// TIA Portal V18 export
// export: Created 2026-01-09T11:31:57.3502958Z, ExportSetting WithDefaults, DisplayName Totally Integrated Automation Portal, DisplayVersion V18 Update 5, DisplayName TIA Portal Openness, DisplayVersion V18 Update 5, DisplayName TIA Portal Teamcenter Gateway, DisplayVersion V18, DisplayName TIA Portal Version Control Interface, DisplayVersion V18, DisplayName SINAMICS Startdrive Advanced, DisplayVersion V18 SP2 Update 1, DisplayName SINAMICS Startdrive G110M, G120, G120C, G120D, G120P, G115D, DisplayVersion V18 SP2 Update 1, DisplayName SINAMICS Startdrive G130, G150, S120, S150, SINAMICS MV, S210, G220, S200, DisplayVersion V18 SP2 Update 1, DisplayName STEP 7 Professional, DisplayVersion V18 Update 5, DisplayName STEP 7 Safety, DisplayVersion V18, DisplayName WinCC Professional, DisplayVersion V18 Update 5
TagTable "Axis"
  Parameter_AxisRun_Axis{1} : ServoType_UDT  (PLC tag Parameter.AxisRun.Axis[1], CPU S71500-2PN_TP700, 1 s)
    TagStructureMember "Pos1"
      TagStructureMember "Position"
      TagStructureMember "Speed"
      TagStructureMember "Reached"
    TagStructureMember "Pos2"
      TagStructureMember "Position"
      TagStructureMember "Speed"
      TagStructureMember "Reached"
    TagStructureMember "Pos3"
      TagStructureMember "Position"
      TagStructureMember "Speed"
      TagStructureMember "Reached"
    TagStructureMember "Pos4"
      TagStructureMember "Position"
      TagStructureMember "Speed"
      TagStructureMember "Reached"
    TagStructureMember "Pos5"
      TagStructureMember "Position"
      TagStructureMember "Speed"
      TagStructureMember "Reached"
    TagStructureMember "Pos6"
      TagStructureMember "Position"
      TagStructureMember "Speed"
      TagStructureMember "Reached"
    TagStructureMember "Pos7"
      TagStructureMember "Position"
      TagStructureMember "Speed"
      TagStructureMember "Reached"
    TagStructureMember "Pos8"
      TagStructureMember "Position"
      TagStructureMember "Speed"
      TagStructureMember "Reached"
    TagStructureMember "Pos9"
      TagStructureMember "Position"
      TagStructureMember "Speed"
      TagStructureMember "Reached"
    TagStructureMember "Pos10"
      TagStructureMember "Position"
      TagStructureMember "Speed"
      TagStructureMember "Reached"
    TagStructureMember "Pos11"
      TagStructureMember "Position"
      TagStructureMember "Speed"
      TagStructureMember "Reached"
    TagStructureMember "Pos12"
      TagStructureMember "Position"
      TagStructureMember "Speed"
      TagStructureMember "Reached"
    TagStructureMember "Pos13"
      TagStructureMember "Position"
      TagStructureMember "Speed"
      TagStructureMember "Reached"
    TagStructureMember "Pos14"
      TagStructureMember "Position"
      TagStructureMember "Speed"
      TagStructureMember "Reached"
    TagStructureMember "Pos15"
      TagStructureMember "Position"
      TagStructureMember "Speed"
      TagStructureMember "Reached"
    TagStructureMember "Pos16"
      TagStructureMember "Position"
      TagStructureMember "Speed"
      TagStructureMember "Reached"
    TagStructureMember "Pos17"
      TagStructureMember "Position"
      TagStructureMember "Speed"
      TagStructureMember "Reached"
    TagStructureMember "Pos18"
      TagStructureMember "Position"
      TagStructureMember "Speed"
      TagStructureMember "Reached"
    TagStructureMember "Pos19"
      TagStructureMember "Position"
      TagStructureMember "Speed"
      TagStructureMember "Reached"
    TagStructureMember "Pos20"
      TagStructureMember "Position"
      TagStructureMember "Speed"
      TagStructureMember "Reached"
    TagStructureMember "Pos21"
      TagStructureMember "Position"
      TagStructureMember "Speed"
      TagStructureMember "Reached"
    TagStructureMember "Pos22"
      TagStructureMember "Position"
      TagStructureMember "Speed"
      TagStructureMember "Reached"
    TagStructureMember "Pos23"
      TagStructureMember "Position"
      TagStructureMember "Speed"
      TagStructureMember "Reached"
    TagStructureMember "Pos24"
      TagStructureMember "Position"
      TagStructureMember "Speed"
      TagStructureMember "Reached"
    TagStructureMember "Pos25"
      TagStructureMember "Position"
      TagStructureMember "Speed"
      TagStructureMember "Reached"
    TagStructureMember "Pos26"
      TagStructureMember "Position"
      TagStructureMember "Speed"
      TagStructureMember "Reached"
    TagStructureMember "Pos27"
      TagStructureMember "Position"
      TagStructureMember "Speed"
      TagStructureMember "Reached"
    TagStructureMember "Pos28"
      TagStructureMember "Position"
      TagStructureMember "Speed"
      TagStructureMember "Reached"
    TagStructureMember "Pos29"
      TagStructureMember "Position"
      TagStructureMember "Speed"
      TagStructureMember "Reached"
    TagStructureMember "Pos30"
      TagStructureMember "Position"
      TagStructureMember "Speed"
      TagStructureMember "Reached"
  Parameter_AxisRun_Axis{2} : ServoType_UDT  (PLC tag Parameter.AxisRun.Axis[2], CPU S71500-2PN_TP700, 1 s)
    TagStructureMember "Pos1"
      TagStructureMember "Position"
      TagStructureMember "Speed"
      TagStructureMember "Reached"
    TagStructureMember "Pos2"
      TagStructureMember "Position"
      TagStructureMember "Speed"
      TagStructureMember "Reached"
    TagStructureMember "Pos3"
      TagStructureMember "Position"
      TagStructureMember "Speed"
      TagStructureMember "Reached"
    TagStructureMember "Pos4"
      TagStructureMember "Position"
      TagStructureMember "Speed"
      TagStructureMember "Reached"
    TagStructureMember "Pos5"
      TagStructureMember "Position"
      TagStructureMember "Speed"
      TagStructureMember "Reached"
    TagStructureMember "Pos6"
      TagStructureMember "Position"
      TagStructureMember "Speed"
      TagStructureMember "Reached"
    TagStructureMember "Pos7"
      TagStructureMember "Position"
      TagStructureMember "Speed"
      TagStructureMember "Reached"
    TagStructureMember "Pos8"
      TagStructureMember "Position"
      TagStructureMember "Speed"
      TagStructureMember "Reached"
    TagStructureMember "Pos9"
      TagStructureMember "Position"
      TagStructureMember "Speed"
      TagStructureMember "Reached"
    TagStructureMember "Pos10"
      TagStructureMember "Position"
      TagStructureMember "Speed"
      TagStructureMember "Reached"
    TagStructureMember "Pos11"
      TagStructureMember "Position"
      TagStructureMember "Speed"
      TagStructureMember "Reached"
    TagStructureMember "Pos12"
      TagStructureMember "Position"
      TagStructureMember "Speed"
      TagStructureMember "Reached"
    TagStructureMember "Pos13"
      TagStructureMember "Position"
      TagStructureMember "Speed"
      TagStructureMember "Reached"
    TagStructureMember "Pos14"
      TagStructureMember "Position"
      TagStructureMember "Speed"
      TagStructureMember "Reached"
    TagStructureMember "Pos15"
      TagStructureMember "Position"
      TagStructureMember "Speed"
      TagStructureMember "Reached"
    TagStructureMember "Pos16"
      TagStructureMember "Position"
      TagStructureMember "Speed"
      TagStructureMember "Reached"
    TagStructureMember "Pos17"
      TagStructureMember "Position"
      TagStructureMember "Speed"
      TagStructureMember "Reached"
    TagStructureMember "Pos18"
      TagStructureMember "Position"
      TagStructureMember "Speed"
      TagStructureMember "Reached"
    TagStructureMember "Pos19"
      TagStructureMember "Position"
      TagStructureMember "Speed"
      TagStructureMember "Reached"
    TagStructureMember "Pos20"
      TagStructureMember "Position"
      TagStructureMember "Speed"
      TagStructureMember "Reached"
    TagStructureMember "Pos21"
      TagStructureMember "Position"
      TagStructureMember "Speed"
      TagStructureMember "Reached"
    TagStructureMember "Pos22"
      TagStructureMember "Position"
      TagStructureMember "Speed"
      TagStructureMember "Reached"
    TagStructureMember "Pos23"
      TagStructureMember "Position"
      TagStructureMember "Speed"
      TagStructureMember "Reached"
    TagStructureMember "Pos24"
      TagStructureMember "Position"
      TagStructureMember "Speed"
      TagStructureMember "Reached"
    TagStructureMember "Pos25"
      TagStructureMember "Position"
      TagStructureMember "Speed"
      TagStructureMember "Reached"
    TagStructureMember "Pos26"
      TagStructureMember "Position"
      TagStructureMember "Speed"
      TagStructureMember "Reached"
    TagStructureMember "Pos27"
      TagStructureMember "Position"
      TagStructureMember "Speed"
      TagStructureMember "Reached"
    TagStructureMember "Pos28"
      TagStructureMember "Position"
      TagStructureMember "Speed"
      TagStructureMember "Reached"
    TagStructureMember "Pos29"
      TagStructureMember "Position"
      TagStructureMember "Speed"
      TagStructureMember "Reached"
    TagStructureMember "Pos30"
      TagStructureMember "Position"
      TagStructureMember "Speed"
      TagStructureMember "Reached"
  Parameter_AxisRun_Axis{3} : ServoType_UDT  (PLC tag Parameter.AxisRun.Axis[3], CPU S71500-2PN_TP700, 1 s)
    TagStructureMember "Pos1"
      TagStructureMember "Position"
      TagStructureMember "Speed"
      TagStructureMember "Reached"
    TagStructureMember "Pos2"
      TagStructureMember "Position"
      TagStructureMember "Speed"
      TagStructureMember "Reached"
    TagStructureMember "Pos3"
      TagStructureMember "Position"
      TagStructureMember "Speed"
      TagStructureMember "Reached"
    TagStructureMember "Pos4"
      TagStructureMember "Position"
      TagStructureMember "Speed"
      TagStructureMember "Reached"
    TagStructureMember "Pos5"
      TagStructureMember "Position"
      TagStructureMember "Speed"
      TagStructureMember "Reached"
    TagStructureMember "Pos6"
      TagStructureMember "Position"
      TagStructureMember "Speed"
      TagStructureMember "Reached"
    TagStructureMember "Pos7"
      TagStructureMember "Position"
      TagStructureMember "Speed"
      TagStructureMember "Reached"
    TagStructureMember "Pos8"
      TagStructureMember "Position"
      TagStructureMember "Speed"
      TagStructureMember "Reached"
    TagStructureMember "Pos9"
      TagStructureMember "Position"
      TagStructureMember "Speed"
      TagStructureMember "Reached"
    TagStructureMember "Pos10"
      TagStructureMember "Position"
      TagStructureMember "Speed"
      TagStructureMember "Reached"
    TagStructureMember "Pos11"
      TagStructureMember "Position"
      TagStructureMember "Speed"
      TagStructureMember "Reached"
    TagStructureMember "Pos12"
      TagStructureMember "Position"
      TagStructureMember "Speed"
      TagStructureMember "Reached"
    TagStructureMember "Pos13"
      TagStructureMember "Position"
      TagStructureMember "Speed"
      TagStructureMember "Reached"
    TagStructureMember "Pos14"
      TagStructureMember "Position"
      TagStructureMember "Speed"
      TagStructureMember "Reached"
    TagStructureMember "Pos15"
      TagStructureMember "Position"
      TagStructureMember "Speed"
      TagStructureMember "Reached"
    TagStructureMember "Pos16"
      TagStructureMember "Position"
      TagStructureMember "Speed"
      TagStructureMember "Reached"
    TagStructureMember "Pos17"
      TagStructureMember "Position"
      TagStructureMember "Speed"
      TagStructureMember "Reached"
    TagStructureMember "Pos18"
      TagStructureMember "Position"
      TagStructureMember "Speed"
      TagStructureMember "Reached"
    TagStructureMember "Pos19"
      TagStructureMember "Position"
      TagStructureMember "Speed"
      TagStructureMember "Reached"
    TagStructureMember "Pos20"
      TagStructureMember "Position"
      TagStructureMember "Speed"
      TagStructureMember "Reached"
    TagStructureMember "Pos21"
      TagStructureMember "Position"
      TagStructureMember "Speed"
      TagStructureMember "Reached"
    TagStructureMember "Pos22"
      TagStructureMember "Position"
      TagStructureMember "Speed"
      TagStructureMember "Reached"
    TagStructureMember "Pos23"
      TagStructureMember "Position"
      TagStructureMember "Speed"
      TagStructureMember "Reached"
    TagStructureMember "Pos24"
      TagStructureMember "Position"
      TagStructureMember "Speed"
      TagStructureMember "Reached"
    TagStructureMember "Pos25"
      TagStructureMember "Position"
      TagStructureMember "Speed"
      TagStructureMember "Reached"
    TagStructureMember "Pos26"
      TagStructureMember "Position"
      TagStructureMember "Speed"
      TagStructureMember "Reached"
    TagStructureMember "Pos27"
      TagStructureMember "Position"
      TagStructureMember "Speed"
      TagStructureMember "Reached"
    TagStructureMember "Pos28"
      TagStructureMember "Position"
      TagStructureMember "Speed"
      TagStructureMember "Reached"
    TagStructureMember "Pos29"
      TagStructureMember "Position"
      TagStructureMember "Speed"
      TagStructureMember "Reached"
    TagStructureMember "Pos30"
      TagStructureMember "Position"
      TagStructureMember "Speed"
      TagStructureMember "Reached"
  Parameter_AxisRun_Axis{4} : ServoType_UDT  (PLC tag Parameter.AxisRun.Axis[4], CPU S71500-2PN_TP700, 1 s)
    TagStructureMember "Pos1"
      TagStructureMember "Position"
      TagStructureMember "Speed"
      TagStructureMember "Reached"
    TagStructureMember "Pos2"
      TagStructureMember "Position"
      TagStructureMember "Speed"
      TagStructureMember "Reached"
    TagStructureMember "Pos3"
      TagStructureMember "Position"
      TagStructureMember "Speed"
      TagStructureMember "Reached"
    TagStructureMember "Pos4"
      TagStructureMember "Position"
      TagStructureMember "Speed"
      TagStructureMember "Reached"
    TagStructureMember "Pos5"
      TagStructureMember "Position"
      TagStructureMember "Speed"
      TagStructureMember "Reached"
    TagStructureMember "Pos6"
      TagStructureMember "Position"
      TagStructureMember "Speed"
      TagStructureMember "Reached"
    TagStructureMember "Pos7"
      TagStructureMember "Position"
      TagStructureMember "Speed"
      TagStructureMember "Reached"
    TagStructureMember "Pos8"
      TagStructureMember "Position"
      TagStructureMember "Speed"
      TagStructureMember "Reached"
    TagStructureMember "Pos9"
      TagStructureMember "Position"
      TagStructureMember "Speed"
      TagStructureMember "Reached"
    TagStructureMember "Pos10"
      TagStructureMember "Position"
      TagStructureMember "Speed"
      TagStructureMember "Reached"
    TagStructureMember "Pos11"
      TagStructureMember "Position"
      TagStructureMember "Speed"
      TagStructureMember "Reached"
    TagStructureMember "Pos12"
      TagStructureMember "Position"
      TagStructureMember "Speed"
      TagStructureMember "Reached"
    TagStructureMember "Pos13"
      TagStructureMember "Position"
      TagStructureMember "Speed"
      TagStructureMember "Reached"
    TagStructureMember "Pos14"
      TagStructureMember "Position"
      TagStructureMember "Speed"
      TagStructureMember "Reached"
    TagStructureMember "Pos15"
      TagStructureMember "Position"
      TagStructureMember "Speed"
      TagStructureMember "Reached"
    TagStructureMember "Pos16"
      TagStructureMember "Position"
      TagStructureMember "Speed"
      TagStructureMember "Reached"
    TagStructureMember "Pos17"
      TagStructureMember "Position"
      TagStructureMember "Speed"
      TagStructureMember "Reached"
    TagStructureMember "Pos18"
      TagStructureMember "Position"
      TagStructureMember "Speed"
      TagStructureMember "Reached"
    TagStructureMember "Pos19"
      TagStructureMember "Position"
      TagStructureMember "Speed"
      TagStructureMember "Reached"
    TagStructureMember "Pos20"
      TagStructureMember "Position"
      TagStructureMember "Speed"
      TagStructureMember "Reached"
    TagStructureMember "Pos21"
      TagStructureMember "Position"
      TagStructureMember "Speed"
      TagStructureMember "Reached"
    TagStructureMember "Pos22"
      TagStructureMember "Position"
      TagStructureMember "Speed"
      TagStructureMember "Reached"
    TagStructureMember "Pos23"
      TagStructureMember "Position"
      TagStructureMember "Speed"
      TagStructureMember "Reached"
    TagStructureMember "Pos24"
      TagStructureMember "Position"
      TagStructureMember "Speed"
      TagStructureMember "Reached"
    TagStructureMember "Pos25"
      TagStructureMember "Position"
      TagStructureMember "Speed"
      TagStructureMember "Reached"
    TagStructureMember "Pos26"
      TagStructureMember "Position"
      TagStructureMember "Speed"
      TagStructureMember "Reached"
    TagStructureMember "Pos27"
      TagStructureMember "Position"
      TagStructureMember "Speed"
      TagStructureMember "Reached"
    TagStructureMember "Pos28"
      TagStructureMember "Position"
      TagStructureMember "Speed"
      TagStructureMember "Reached"
    TagStructureMember "Pos29"
      TagStructureMember "Position"
      TagStructureMember "Speed"
      TagStructureMember "Reached"
    TagStructureMember "Pos30"
      TagStructureMember "Position"
      TagStructureMember "Speed"
      TagStructureMember "Reached"
  Parameter_AxisRun_Axis{5} : ServoType_UDT  (PLC tag Parameter.AxisRun.Axis[5], CPU S71500-2PN_TP700, 1 s)
    TagStructureMember "Pos1"
      TagStructureMember "Position"
      TagStructureMember "Speed"
      TagStructureMember "Reached"
    TagStructureMember "Pos2"
      TagStructureMember "Position"
      TagStructureMember "Speed"
      TagStructureMember "Reached"
    TagStructureMember "Pos3"
      TagStructureMember "Position"
      TagStructureMember "Speed"
      TagStructureMember "Reached"
    TagStructureMember "Pos4"
      TagStructureMember "Position"
      TagStructureMember "Speed"
      TagStructureMember "Reached"
    TagStructureMember "Pos5"
      TagStructureMember "Position"
      TagStructureMember "Speed"
      TagStructureMember "Reached"
    TagStructureMember "Pos6"
      TagStructureMember "Position"
      TagStructureMember "Speed"
      TagStructureMember "Reached"
    TagStructureMember "Pos7"
      TagStructureMember "Position"
      TagStructureMember "Speed"
      TagStructureMember "Reached"
    TagStructureMember "Pos8"
      TagStructureMember "Position"
      TagStructureMember "Speed"
      TagStructureMember "Reached"
    TagStructureMember "Pos9"
      TagStructureMember "Position"
      TagStructureMember "Speed"
      TagStructureMember "Reached"
    TagStructureMember "Pos10"
      TagStructureMember "Position"
      TagStructureMember "Speed"
      TagStructureMember "Reached"
    TagStructureMember "Pos11"
      TagStructureMember "Position"
      TagStructureMember "Speed"
      TagStructureMember "Reached"
    TagStructureMember "Pos12"
      TagStructureMember "Position"
      TagStructureMember "Speed"
      TagStructureMember "Reached"
    TagStructureMember "Pos13"
      TagStructureMember "Position"
      TagStructureMember "Speed"
      TagStructureMember "Reached"
    TagStructureMember "Pos14"
      TagStructureMember "Position"
      TagStructureMember "Speed"
      TagStructureMember "Reached"
    TagStructureMember "Pos15"
      TagStructureMember "Position"
      TagStructureMember "Speed"
      TagStructureMember "Reached"
    TagStructureMember "Pos16"
      TagStructureMember "Position"
      TagStructureMember "Speed"
      TagStructureMember "Reached"
    TagStructureMember "Pos17"
      TagStructureMember "Position"
      TagStructureMember "Speed"
      TagStructureMember "Reached"
    TagStructureMember "Pos18"
      TagStructureMember "Position"
      TagStructureMember "Speed"
      TagStructureMember "Reached"
    TagStructureMember "Pos19"
      TagStructureMember "Position"
      TagStructureMember "Speed"
      TagStructureMember "Reached"
    TagStructureMember "Pos20"
      TagStructureMember "Position"
      TagStructureMember "Speed"
      TagStructureMember "Reached"
    TagStructureMember "Pos21"
      TagStructureMember "Position"
      TagStructureMember "Speed"
      TagStructureMember "Reached"
    TagStructureMember "Pos22"
      TagStructureMember "Position"
      TagStructureMember "Speed"
      TagStructureMember "Reached"
    TagStructureMember "Pos23"
      TagStructureMember "Position"
      TagStructureMember "Speed"
      TagStructureMember "Reached"
    TagStructureMember "Pos24"
      TagStructureMember "Position"
      TagStructureMember "Speed"
      TagStructureMember "Reached"
    TagStructureMember "Pos25"
      TagStructureMember "Position"
      TagStructureMember "Speed"
      TagStructureMember "Reached"
    TagStructureMember "Pos26"
      TagStructureMember "Position"
      TagStructureMember "Speed"
      TagStructureMember "Reached"
    TagStructureMember "Pos27"
      TagStructureMember "Position"
      TagStructureMember "Speed"
      TagStructureMember "Reached"
    TagStructureMember "Pos28"
      TagStructureMember "Position"
      TagStructureMember "Speed"
      TagStructureMember "Reached"
    TagStructureMember "Pos29"
      TagStructureMember "Position"
      TagStructureMember "Speed"
      TagStructureMember "Reached"
    TagStructureMember "Pos30"
      TagStructureMember "Position"
      TagStructureMember "Speed"
      TagStructureMember "Reached"
  Parameter_AxisRun_Axis{6} : ServoType_UDT  (PLC tag Parameter.AxisRun.Axis[6], CPU S71500-2PN_TP700, 1 s)
    TagStructureMember "Pos1"
      TagStructureMember "Position"
      TagStructureMember "Speed"
      TagStructureMember "Reached"
    TagStructureMember "Pos2"
      TagStructureMember "Position"
      TagStructureMember "Speed"
      TagStructureMember "Reached"
    TagStructureMember "Pos3"
      TagStructureMember "Position"
      TagStructureMember "Speed"
      TagStructureMember "Reached"
    TagStructureMember "Pos4"
      TagStructureMember "Position"
      TagStructureMember "Speed"
      TagStructureMember "Reached"
    TagStructureMember "Pos5"
      TagStructureMember "Position"
      TagStructureMember "Speed"
      TagStructureMember "Reached"
    TagStructureMember "Pos6"
      TagStructureMember "Position"
      TagStructureMember "Speed"
      TagStructureMember "Reached"
    TagStructureMember "Pos7"
      TagStructureMember "Position"
      TagStructureMember "Speed"
      TagStructureMember "Reached"
    TagStructureMember "Pos8"
      TagStructureMember "Position"
      TagStructureMember "Speed"
      TagStructureMember "Reached"
    TagStructureMember "Pos9"
      TagStructureMember "Position"
      TagStructureMember "Speed"
      TagStructureMember "Reached"
    TagStructureMember "Pos10"
      TagStructureMember "Position"
      TagStructureMember "Speed"
      TagStructureMember "Reached"
    TagStructureMember "Pos11"
      TagStructureMember "Position"
      TagStructureMember "Speed"
      TagStructureMember "Reached"
    TagStructureMember "Pos12"
      TagStructureMember "Position"
      TagStructureMember "Speed"
      TagStructureMember "Reached"
    TagStructureMember "Pos13"
      TagStructureMember "Position"
      TagStructureMember "Speed"
      TagStructureMember "Reached"
    TagStructureMember "Pos14"
      TagStructureMember "Position"
      TagStructureMember "Speed"
      TagStructureMember "Reached"
    TagStructureMember "Pos15"
      TagStructureMember "Position"
      TagStructureMember "Speed"
      TagStructureMember "Reached"
    TagStructureMember "Pos16"
      TagStructureMember "Position"
      TagStructureMember "Speed"
      TagStructureMember "Reached"
    TagStructureMember "Pos17"
      TagStructureMember "Position"
      TagStructureMember "Speed"
      TagStructureMember "Reached"
    TagStructureMember "Pos18"
      TagStructureMember "Position"
      TagStructureMember "Speed"
      TagStructureMember "Reached"
    TagStructureMember "Pos19"
      TagStructureMember "Position"
      TagStructureMember "Speed"
      TagStructureMember "Reached"
    TagStructureMember "Pos20"
      TagStructureMember "Position"
      TagStructureMember "Speed"
      TagStructureMember "Reached"
    TagStructureMember "Pos21"
      TagStructureMember "Position"
      TagStructureMember "Speed"
      TagStructureMember "Reached"
    TagStructureMember "Pos22"
      TagStructureMember "Position"
      TagStructureMember "Speed"
      TagStructureMember "Reached"
    TagStructureMember "Pos23"
      TagStructureMember "Position"
      TagStructureMember "Speed"
      TagStructureMember "Reached"
    TagStructureMember "Pos24"
      TagStructureMember "Position"
      TagStructureMember "Speed"
      TagStructureMember "Reached"
    TagStructureMember "Pos25"
      TagStructureMember "Position"
      TagStructureMember "Speed"
      TagStructureMember "Reached"
    TagStructureMember "Pos26"
      TagStructureMember "Position"
      TagStructureMember "Speed"
      TagStructureMember "Reached"
    TagStructureMember "Pos27"
      TagStructureMember "Position"
      TagStructureMember "Speed"
      TagStructureMember "Reached"
    TagStructureMember "Pos28"
      TagStructureMember "Position"
      TagStructureMember "Speed"
      TagStructureMember "Reached"
    TagStructureMember "Pos29"
      TagStructureMember "Position"
      TagStructureMember "Speed"
      TagStructureMember "Reached"
    TagStructureMember "Pos30"
      TagStructureMember "Position"
      TagStructureMember "Speed"
      TagStructureMember "Reached"
  Parameter_AxisRun_Axis{7} : ServoType_UDT  (PLC tag Parameter.AxisRun.Axis[7], CPU S71500-2PN_TP700, 1 s)
    TagStructureMember "Pos1"
      TagStructureMember "Position"
      TagStructureMember "Speed"
      TagStructureMember "Reached"
    TagStructureMember "Pos2"
      TagStructureMember "Position"
      TagStructureMember "Speed"
      TagStructureMember "Reached"
    TagStructureMember "Pos3"
      TagStructureMember "Position"
      TagStructureMember "Speed"
      TagStructureMember "Reached"
    TagStructureMember "Pos4"
      TagStructureMember "Position"
      TagStructureMember "Speed"
      TagStructureMember "Reached"
    TagStructureMember "Pos5"
      TagStructureMember "Position"
      TagStructureMember "Speed"
      TagStructureMember "Reached"
    TagStructureMember "Pos6"
      TagStructureMember "Position"
      TagStructureMember "Speed"
      TagStructureMember "Reached"
    TagStructureMember "Pos7"
      TagStructureMember "Position"
      TagStructureMember "Speed"
      TagStructureMember "Reached"
    TagStructureMember "Pos8"
      TagStructureMember "Position"
      TagStructureMember "Speed"
      TagStructureMember "Reached"
    TagStructureMember "Pos9"
      TagStructureMember "Position"
      TagStructureMember "Speed"
      TagStructureMember "Reached"
    TagStructureMember "Pos10"
      TagStructureMember "Position"
      TagStructureMember "Speed"
      TagStructureMember "Reached"
    TagStructureMember "Pos11"
      TagStructureMember "Position"
      TagStructureMember "Speed"
      TagStructureMember "Reached"
    TagStructureMember "Pos12"
      TagStructureMember "Position"
      TagStructureMember "Speed"
      TagStructureMember "Reached"
    TagStructureMember "Pos13"
      TagStructureMember "Position"
      TagStructureMember "Speed"
      TagStructureMember "Reached"
    TagStructureMember "Pos14"
      TagStructureMember "Position"
      TagStructureMember "Speed"
      TagStructureMember "Reached"
    TagStructureMember "Pos15"
      TagStructureMember "Position"
      TagStructureMember "Speed"
      TagStructureMember "Reached"
    TagStructureMember "Pos16"
      TagStructureMember "Position"
      TagStructureMember "Speed"
      TagStructureMember "Reached"
    TagStructureMember "Pos17"
      TagStructureMember "Position"
      TagStructureMember "Speed"
      TagStructureMember "Reached"
    TagStructureMember "Pos18"
      TagStructureMember "Position"
      TagStructureMember "Speed"
      TagStructureMember "Reached"
    TagStructureMember "Pos19"
      TagStructureMember "Position"
      TagStructureMember "Speed"
      TagStructureMember "Reached"
    TagStructureMember "Pos20"
      TagStructureMember "Position"
      TagStructureMember "Speed"
      TagStructureMember "Reached"
    TagStructureMember "Pos21"
      TagStructureMember "Position"
      TagStructureMember "Speed"
      TagStructureMember "Reached"
    TagStructureMember "Pos22"
      TagStructureMember "Position"
      TagStructureMember "Speed"
      TagStructureMember "Reached"
    TagStructureMember "Pos23"
      TagStructureMember "Position"
      TagStructureMember "Speed"
      TagStructureMember "Reached"
    TagStructureMember "Pos24"
      TagStructureMember "Position"
      TagStructureMember "Speed"
      TagStructureMember "Reached"
    TagStructureMember "Pos25"
      TagStructureMember "Position"
      TagStructureMember "Speed"
      TagStructureMember "Reached"
    TagStructureMember "Pos26"
      TagStructureMember "Position"
      TagStructureMember "Speed"
      TagStructureMember "Reached"
    TagStructureMember "Pos27"
      TagStructureMember "Position"
      TagStructureMember "Speed"
      TagStructureMember "Reached"
    TagStructureMember "Pos28"
      TagStructureMember "Position"
      TagStructureMember "Speed"
      TagStructureMember "Reached"
    TagStructureMember "Pos29"
      TagStructureMember "Position"
      TagStructureMember "Speed"
      TagStructureMember "Reached"
    TagStructureMember "Pos30"
      TagStructureMember "Position"
      TagStructureMember "Speed"
      TagStructureMember "Reached"
  Parameter_AxisRun_Axis{8} : ServoType_UDT  (PLC tag Parameter.AxisRun.Axis[8], CPU S71500-2PN_TP700, 1 s)
    TagStructureMember "Pos1"
      TagStructureMember "Position"
      TagStructureMember "Speed"
      TagStructureMember "Reached"
    TagStructureMember "Pos2"
      TagStructureMember "Position"
      TagStructureMember "Speed"
      TagStructureMember "Reached"
    TagStructureMember "Pos3"
      TagStructureMember "Position"
      TagStructureMember "Speed"
      TagStructureMember "Reached"
    TagStructureMember "Pos4"
      TagStructureMember "Position"
      TagStructureMember "Speed"
      TagStructureMember "Reached"
    TagStructureMember "Pos5"
      TagStructureMember "Position"
      TagStructureMember "Speed"
      TagStructureMember "Reached"
    TagStructureMember "Pos6"
      TagStructureMember "Position"
      TagStructureMember "Speed"
      TagStructureMember "Reached"
    TagStructureMember "Pos7"
      TagStructureMember "Position"
      TagStructureMember "Speed"
      TagStructureMember "Reached"
    TagStructureMember "Pos8"
      TagStructureMember "Position"
      TagStructureMember "Speed"
      TagStructureMember "Reached"
    TagStructureMember "Pos9"
      TagStructureMember "Position"
      TagStructureMember "Speed"
      TagStructureMember "Reached"
    TagStructureMember "Pos10"
      TagStructureMember "Position"
      TagStructureMember "Speed"
      TagStructureMember "Reached"
    TagStructureMember "Pos11"
      TagStructureMember "Position"
      TagStructureMember "Speed"
      TagStructureMember "Reached"
    TagStructureMember "Pos12"
      TagStructureMember "Position"
      TagStructureMember "Speed"
      TagStructureMember "Reached"
    TagStructureMember "Pos13"
      TagStructureMember "Position"
      TagStructureMember "Speed"
      TagStructureMember "Reached"
    TagStructureMember "Pos14"
      TagStructureMember "Position"
      TagStructureMember "Speed"
      TagStructureMember "Reached"
    TagStructureMember "Pos15"
      TagStructureMember "Position"
      TagStructureMember "Speed"
      TagStructureMember "Reached"
    TagStructureMember "Pos16"
      TagStructureMember "Position"
      TagStructureMember "Speed"
      TagStructureMember "Reached"
    TagStructureMember "Pos17"
      TagStructureMember "Position"
      TagStructureMember "Speed"
      TagStructureMember "Reached"
    TagStructureMember "Pos18"
      TagStructureMember "Position"
      TagStructureMember "Speed"
      TagStructureMember "Reached"
    TagStructureMember "Pos19"
      TagStructureMember "Position"
      TagStructureMember "Speed"
      TagStructureMember "Reached"
    TagStructureMember "Pos20"
      TagStructureMember "Position"
      TagStructureMember "Speed"
      TagStructureMember "Reached"
    TagStructureMember "Pos21"
      TagStructureMember "Position"
      TagStructureMember "Speed"
      TagStructureMember "Reached"
    TagStructureMember "Pos22"
      TagStructureMember "Position"
      TagStructureMember "Speed"
      TagStructureMember "Reached"
    TagStructureMember "Pos23"
      TagStructureMember "Position"
      TagStructureMember "Speed"
      TagStructureMember "Reached"
    TagStructureMember "Pos24"
      TagStructureMember "Position"
      TagStructureMember "Speed"
      TagStructureMember "Reached"
    TagStructureMember "Pos25"
      TagStructureMember "Position"
      TagStructureMember "Speed"
      TagStructureMember "Reached"
    TagStructureMember "Pos26"
      TagStructureMember "Position"
      TagStructureMember "Speed"
      TagStructureMember "Reached"
    TagStructureMember "Pos27"
      TagStructureMember "Position"
      TagStructureMember "Speed"
      TagStructureMember "Reached"
    TagStructureMember "Pos28"
      TagStructureMember "Position"
      TagStructureMember "Speed"
      TagStructureMember "Reached"
    TagStructureMember "Pos29"
      TagStructureMember "Position"
      TagStructureMember "Speed"
      TagStructureMember "Reached"
    TagStructureMember "Pos30"
      TagStructureMember "Position"
      TagStructureMember "Speed"
      TagStructureMember "Reached"
  Parameter_AxisRun_Axis{9} : ServoType_UDT  (PLC tag Parameter.AxisRun.Axis[9], CPU S71500-2PN_TP700, 1 s)
    TagStructureMember "Pos1"
      TagStructureMember "Position"
      TagStructureMember "Speed"
      TagStructureMember "Reached"
    TagStructureMember "Pos2"
      TagStructureMember "Position"
      TagStructureMember "Speed"
      TagStructureMember "Reached"
    TagStructureMember "Pos3"
      TagStructureMember "Position"
      TagStructureMember "Speed"
      TagStructureMember "Reached"
    TagStructureMember "Pos4"
      TagStructureMember "Position"
      TagStructureMember "Speed"
      TagStructureMember "Reached"
    TagStructureMember "Pos5"
      TagStructureMember "Position"
      TagStructureMember "Speed"
      TagStructureMember "Reached"
    TagStructureMember "Pos6"
      TagStructureMember "Position"
      TagStructureMember "Speed"
      TagStructureMember "Reached"
    TagStructureMember "Pos7"
      TagStructureMember "Position"
      TagStructureMember "Speed"
      TagStructureMember "Reached"
    TagStructureMember "Pos8"
      TagStructureMember "Position"
      TagStructureMember "Speed"
      TagStructureMember "Reached"
    TagStructureMember "Pos9"
      TagStructureMember "Position"
      TagStructureMember "Speed"
      TagStructureMember "Reached"
    TagStructureMember "Pos10"
      TagStructureMember "Position"
      TagStructureMember "Speed"
      TagStructureMember "Reached"
    TagStructureMember "Pos11"
      TagStructureMember "Position"
      TagStructureMember "Speed"
      TagStructureMember "Reached"
    TagStructureMember "Pos12"
      TagStructureMember "Position"
      TagStructureMember "Speed"
      TagStructureMember "Reached"
    TagStructureMember "Pos13"
      TagStructureMember "Position"
      TagStructureMember "Speed"
      TagStructureMember "Reached"
    TagStructureMember "Pos14"
      TagStructureMember "Position"
      TagStructureMember "Speed"
      TagStructureMember "Reached"
    TagStructureMember "Pos15"
      TagStructureMember "Position"
      TagStructureMember "Speed"
      TagStructureMember "Reached"
    TagStructureMember "Pos16"
      TagStructureMember "Position"
      TagStructureMember "Speed"
      TagStructureMember "Reached"
    TagStructureMember "Pos17"
      TagStructureMember "Position"
      TagStructureMember "Speed"
      TagStructureMember "Reached"
    TagStructureMember "Pos18"
      TagStructureMember "Position"
      TagStructureMember "Speed"
      TagStructureMember "Reached"
    TagStructureMember "Pos19"
      TagStructureMember "Position"
      TagStructureMember "Speed"
      TagStructureMember "Reached"
    TagStructureMember "Pos20"
      TagStructureMember "Position"
      TagStructureMember "Speed"
      TagStructureMember "Reached"
    TagStructureMember "Pos21"
      TagStructureMember "Position"
      TagStructureMember "Speed"
      TagStructureMember "Reached"
    TagStructureMember "Pos22"
      TagStructureMember "Position"
      TagStructureMember "Speed"
      TagStructureMember "Reached"
    TagStructureMember "Pos23"
      TagStructureMember "Position"
      TagStructureMember "Speed"
      TagStructureMember "Reached"
    TagStructureMember "Pos24"
      TagStructureMember "Position"
      TagStructureMember "Speed"
      TagStructureMember "Reached"
    TagStructureMember "Pos25"
      TagStructureMember "Position"
      TagStructureMember "Speed"
      TagStructureMember "Reached"
    TagStructureMember "Pos26"
      TagStructureMember "Position"
      TagStructureMember "Speed"
      TagStructureMember "Reached"
    TagStructureMember "Pos27"
      TagStructureMember "Position"
      TagStructureMember "Speed"
      TagStructureMember "Reached"
    TagStructureMember "Pos28"
      TagStructureMember "Position"
      TagStructureMember "Speed"
      TagStructureMember "Reached"
    TagStructureMember "Pos29"
      TagStructureMember "Position"
      TagStructureMember "Speed"
      TagStructureMember "Reached"
    TagStructureMember "Pos30"
      TagStructureMember "Position"
      TagStructureMember "Speed"
      TagStructureMember "Reached"
  Parameter_AxisRun_Axis{10} : ServoType_UDT  (PLC tag Parameter.AxisRun.Axis[10], CPU S71500-2PN_TP700, 1 s)
    TagStructureMember "Pos1"
      TagStructureMember "Position"
      TagStructureMember "Speed"
      TagStructureMember "Reached"
    TagStructureMember "Pos2"
      TagStructureMember "Position"
      TagStructureMember "Speed"
      TagStructureMember "Reached"
    TagStructureMember "Pos3"
      TagStructureMember "Position"
      TagStructureMember "Speed"
      TagStructureMember "Reached"
    TagStructureMember "Pos4"
      TagStructureMember "Position"
      TagStructureMember "Speed"
      TagStructureMember "Reached"
    TagStructureMember "Pos5"
      TagStructureMember "Position"
      TagStructureMember "Speed"
      TagStructureMember "Reached"
    TagStructureMember "Pos6"
      TagStructureMember "Position"
      TagStructureMember "Speed"
      TagStructureMember "Reached"
    TagStructureMember "Pos7"
      TagStructureMember "Position"
      TagStructureMember "Speed"
      TagStructureMember "Reached"
    TagStructureMember "Pos8"
      TagStructureMember "Position"
      TagStructureMember "Speed"
      TagStructureMember "Reached"
    TagStructureMember "Pos9"
      TagStructureMember "Position"
      TagStructureMember "Speed"
      TagStructureMember "Reached"
    TagStructureMember "Pos10"
      TagStructureMember "Position"
      TagStructureMember "Speed"
      TagStructureMember "Reached"
    TagStructureMember "Pos11"
      TagStructureMember "Position"
      TagStructureMember "Speed"
      TagStructureMember "Reached"
    TagStructureMember "Pos12"
      TagStructureMember "Position"
      TagStructureMember "Speed"
      TagStructureMember "Reached"
    TagStructureMember "Pos13"
      TagStructureMember "Position"
      TagStructureMember "Speed"
      TagStructureMember "Reached"
    TagStructureMember "Pos14"
      TagStructureMember "Position"
      TagStructureMember "Speed"
      TagStructureMember "Reached"
    TagStructureMember "Pos15"
      TagStructureMember "Position"
      TagStructureMember "Speed"
      TagStructureMember "Reached"
    TagStructureMember "Pos16"
      TagStructureMember "Position"
      TagStructureMember "Speed"
      TagStructureMember "Reached"
    TagStructureMember "Pos17"
      TagStructureMember "Position"
      TagStructureMember "Speed"
      TagStructureMember "Reached"
    TagStructureMember "Pos18"
      TagStructureMember "Position"
      TagStructureMember "Speed"
      TagStructureMember "Reached"
    TagStructureMember "Pos19"
      TagStructureMember "Position"
      TagStructureMember "Speed"
      TagStructureMember "Reached"
    TagStructureMember "Pos20"
      TagStructureMember "Position"
      TagStructureMember "Speed"
      TagStructureMember "Reached"
    TagStructureMember "Pos21"
      TagStructureMember "Position"
      TagStructureMember "Speed"
      TagStructureMember "Reached"
    TagStructureMember "Pos22"
      TagStructureMember "Position"
      TagStructureMember "Speed"
      TagStructureMember "Reached"
    TagStructureMember "Pos23"
      TagStructureMember "Position"
      TagStructureMember "Speed"
      TagStructureMember "Reached"
    TagStructureMember "Pos24"
      TagStructureMember "Position"
      TagStructureMember "Speed"
      TagStructureMember "Reached"
    TagStructureMember "Pos25"
      TagStructureMember "Position"
      TagStructureMember "Speed"
      TagStructureMember "Reached"
    TagStructureMember "Pos26"
      TagStructureMember "Position"
      TagStructureMember "Speed"
      TagStructureMember "Reached"
    TagStructureMember "Pos27"
      TagStructureMember "Position"
      TagStructureMember "Speed"
      TagStructureMember "Reached"
    TagStructureMember "Pos28"
      TagStructureMember "Position"
      TagStructureMember "Speed"
      TagStructureMember "Reached"
    TagStructureMember "Pos29"
      TagStructureMember "Position"
      TagStructureMember "Speed"
      TagStructureMember "Reached"
    TagStructureMember "Pos30"
      TagStructureMember "Position"
      TagStructureMember "Speed"
      TagStructureMember "Reached"
  Parameter_AxisRun_Axis{11} : ServoType_UDT  (PLC tag Parameter.AxisRun.Axis[11], CPU S71500-2PN_TP700, 1 s)
    TagStructureMember "Pos1"
      TagStructureMember "Position"
      TagStructureMember "Speed"
      TagStructureMember "Reached"
    TagStructureMember "Pos2"
      TagStructureMember "Position"
      TagStructureMember "Speed"
      TagStructureMember "Reached"
    TagStructureMember "Pos3"
      TagStructureMember "Position"
      TagStructureMember "Speed"
      TagStructureMember "Reached"
    TagStructureMember "Pos4"
      TagStructureMember "Position"
      TagStructureMember "Speed"
      TagStructureMember "Reached"
    TagStructureMember "Pos5"
      TagStructureMember "Position"
      TagStructureMember "Speed"
      TagStructureMember "Reached"
    TagStructureMember "Pos6"
      TagStructureMember "Position"
      TagStructureMember "Speed"
      TagStructureMember "Reached"
    TagStructureMember "Pos7"
      TagStructureMember "Position"
      TagStructureMember "Speed"
      TagStructureMember "Reached"
    TagStructureMember "Pos8"
      TagStructureMember "Position"
      TagStructureMember "Speed"
      TagStructureMember "Reached"
    TagStructureMember "Pos9"
      TagStructureMember "Position"
      TagStructureMember "Speed"
      TagStructureMember "Reached"
    TagStructureMember "Pos10"
      TagStructureMember "Position"
      TagStructureMember "Speed"
      TagStructureMember "Reached"
    TagStructureMember "Pos11"
      TagStructureMember "Position"
      TagStructureMember "Speed"
      TagStructureMember "Reached"
    TagStructureMember "Pos12"
      TagStructureMember "Position"
      TagStructureMember "Speed"
      TagStructureMember "Reached"
    TagStructureMember "Pos13"
      TagStructureMember "Position"
      TagStructureMember "Speed"
      TagStructureMember "Reached"
    TagStructureMember "Pos14"
      TagStructureMember "Position"
      TagStructureMember "Speed"
      TagStructureMember "Reached"
    TagStructureMember "Pos15"
      TagStructureMember "Position"
      TagStructureMember "Speed"
      TagStructureMember "Reached"
    TagStructureMember "Pos16"
      TagStructureMember "Position"
      TagStructureMember "Speed"
      TagStructureMember "Reached"
    TagStructureMember "Pos17"
      TagStructureMember "Position"
      TagStructureMember "Speed"
      TagStructureMember "Reached"
    TagStructureMember "Pos18"
      TagStructureMember "Position"
      TagStructureMember "Speed"
      TagStructureMember "Reached"
    TagStructureMember "Pos19"
      TagStructureMember "Position"
      TagStructureMember "Speed"
      TagStructureMember "Reached"
    TagStructureMember "Pos20"
      TagStructureMember "Position"
      TagStructureMember "Speed"
      TagStructureMember "Reached"
    TagStructureMember "Pos21"
      TagStructureMember "Position"
      TagStructureMember "Speed"
      TagStructureMember "Reached"
    TagStructureMember "Pos22"
      TagStructureMember "Position"
      TagStructureMember "Speed"
      TagStructureMember "Reached"
    TagStructureMember "Pos23"
      TagStructureMember "Position"
      TagStructureMember "Speed"
      TagStructureMember "Reached"
    TagStructureMember "Pos24"
      TagStructureMember "Position"
      TagStructureMember "Speed"
      TagStructureMember "Reached"
    TagStructureMember "Pos25"
      TagStructureMember "Position"
      TagStructureMember "Speed"
      TagStructureMember "Reached"
    TagStructureMember "Pos26"
      TagStructureMember "Position"
      TagStructureMember "Speed"
      TagStructureMember "Reached"
    TagStructureMember "Pos27"
      TagStructureMember "Position"
      TagStructureMember "Speed"
      TagStructureMember "Reached"
    TagStructureMember "Pos28"
      TagStructureMember "Position"
      TagStructureMember "Speed"
      TagStructureMember "Reached"
    TagStructureMember "Pos29"
      TagStructureMember "Position"
      TagStructureMember "Speed"
      TagStructureMember "Reached"
    TagStructureMember "Pos30"
      TagStructureMember "Position"
      TagStructureMember "Speed"
      TagStructureMember "Reached"
  Parameter_AxisRun_Axis{12} : ServoType_UDT  (PLC tag Parameter.AxisRun.Axis[12], CPU S71500-2PN_TP700, 1 s)
    TagStructureMember "Pos1"
      TagStructureMember "Position"
      TagStructureMember "Speed"
      TagStructureMember "Reached"
    TagStructureMember "Pos2"
      TagStructureMember "Position"
      TagStructureMember "Speed"
      TagStructureMember "Reached"
    TagStructureMember "Pos3"
      TagStructureMember "Position"
      TagStructureMember "Speed"
      TagStructureMember "Reached"
    TagStructureMember "Pos4"
      TagStructureMember "Position"
      TagStructureMember "Speed"
      TagStructureMember "Reached"
    TagStructureMember "Pos5"
      TagStructureMember "Position"
      TagStructureMember "Speed"
      TagStructureMember "Reached"
    TagStructureMember "Pos6"
      TagStructureMember "Position"
      TagStructureMember "Speed"
      TagStructureMember "Reached"
    TagStructureMember "Pos7"
      TagStructureMember "Position"
      TagStructureMember "Speed"
      TagStructureMember "Reached"
    TagStructureMember "Pos8"
      TagStructureMember "Position"
      TagStructureMember "Speed"
      TagStructureMember "Reached"
    TagStructureMember "Pos9"
      TagStructureMember "Position"
      TagStructureMember "Speed"
      TagStructureMember "Reached"
    TagStructureMember "Pos10"
      TagStructureMember "Position"
      TagStructureMember "Speed"
      TagStructureMember "Reached"
    TagStructureMember "Pos11"
      TagStructureMember "Position"
      TagStructureMember "Speed"
      TagStructureMember "Reached"
    TagStructureMember "Pos12"
      TagStructureMember "Position"
      TagStructureMember "Speed"
      TagStructureMember "Reached"
    TagStructureMember "Pos13"
      TagStructureMember "Position"
      TagStructureMember "Speed"
      TagStructureMember "Reached"
    TagStructureMember "Pos14"
      TagStructureMember "Position"
      TagStructureMember "Speed"
      TagStructureMember "Reached"
    TagStructureMember "Pos15"
      TagStructureMember "Position"
      TagStructureMember "Speed"
      TagStructureMember "Reached"
    TagStructureMember "Pos16"
      TagStructureMember "Position"
      TagStructureMember "Speed"
      TagStructureMember "Reached"
    TagStructureMember "Pos17"
      TagStructureMember "Position"
      TagStructureMember "Speed"
      TagStructureMember "Reached"
    TagStructureMember "Pos18"
      TagStructureMember "Position"
      TagStructureMember "Speed"
      TagStructureMember "Reached"
    TagStructureMember "Pos19"
      TagStructureMember "Position"
      TagStructureMember "Speed"
      TagStructureMember "Reached"
    TagStructureMember "Pos20"
      TagStructureMember "Position"
      TagStructureMember "Speed"
      TagStructureMember "Reached"
    TagStructureMember "Pos21"
      TagStructureMember "Position"
      TagStructureMember "Speed"
      TagStructureMember "Reached"
    TagStructureMember "Pos22"
      TagStructureMember "Position"
      TagStructureMember "Speed"
      TagStructureMember "Reached"
    TagStructureMember "Pos23"
      TagStructureMember "Position"
      TagStructureMember "Speed"
      TagStructureMember "Reached"
    TagStructureMember "Pos24"
      TagStructureMember "Position"
      TagStructureMember "Speed"
      TagStructureMember "Reached"
    TagStructureMember "Pos25"
      TagStructureMember "Position"
      TagStructureMember "Speed"
      TagStructureMember "Reached"
    TagStructureMember "Pos26"
      TagStructureMember "Position"
      TagStructureMember "Speed"
      TagStructureMember "Reached"
    TagStructureMember "Pos27"
      TagStructureMember "Position"
      TagStructureMember "Speed"
      TagStructureMember "Reached"
    TagStructureMember "Pos28"
      TagStructureMember "Position"
      TagStructureMember "Speed"
      TagStructureMember "Reached"
    TagStructureMember "Pos29"
      TagStructureMember "Position"
      TagStructureMember "Speed"
      TagStructureMember "Reached"
    TagStructureMember "Pos30"
      TagStructureMember "Position"
      TagStructureMember "Speed"
      TagStructureMember "Reached"
  Parameter_AxisRun_Axis{13} : ServoType_UDT  (PLC tag Parameter.AxisRun.Axis[13], CPU S71500-2PN_TP700, 1 s)
    TagStructureMember "Pos1"
      TagStructureMember "Position"
      TagStructureMember "Speed"
      TagStructureMember "Reached"
    TagStructureMember "Pos2"
      TagStructureMember "Position"
      TagStructureMember "Speed"
      TagStructureMember "Reached"
    TagStructureMember "Pos3"
      TagStructureMember "Position"
      TagStructureMember "Speed"
      TagStructureMember "Reached"
    TagStructureMember "Pos4"
      TagStructureMember "Position"
      TagStructureMember "Speed"
      TagStructureMember "Reached"
    TagStructureMember "Pos5"
      TagStructureMember "Position"
      TagStructureMember "Speed"
      TagStructureMember "Reached"
    TagStructureMember "Pos6"
      TagStructureMember "Position"
      TagStructureMember "Speed"
      TagStructureMember "Reached"
    TagStructureMember "Pos7"
      TagStructureMember "Position"
      TagStructureMember "Speed"
      TagStructureMember "Reached"
    TagStructureMember "Pos8"
      TagStructureMember "Position"
      TagStructureMember "Speed"
      TagStructureMember "Reached"
    TagStructureMember "Pos9"
      TagStructureMember "Position"
      TagStructureMember "Speed"
      TagStructureMember "Reached"
    TagStructureMember "Pos10"
      TagStructureMember "Position"
      TagStructureMember "Speed"
      TagStructureMember "Reached"
    TagStructureMember "Pos11"
      TagStructureMember "Position"
      TagStructureMember "Speed"
      TagStructureMember "Reached"
    TagStructureMember "Pos12"
      TagStructureMember "Position"
      TagStructureMember "Speed"
      TagStructureMember "Reached"
    TagStructureMember "Pos13"
      TagStructureMember "Position"
      TagStructureMember "Speed"
      TagStructureMember "Reached"
    TagStructureMember "Pos14"
      TagStructureMember "Position"
      TagStructureMember "Speed"
      TagStructureMember "Reached"
    TagStructureMember "Pos15"
      TagStructureMember "Position"
      TagStructureMember "Speed"
      TagStructureMember "Reached"
    TagStructureMember "Pos16"
      TagStructureMember "Position"
      TagStructureMember "Speed"
      TagStructureMember "Reached"
    TagStructureMember "Pos17"
      TagStructureMember "Position"
      TagStructureMember "Speed"
      TagStructureMember "Reached"
    TagStructureMember "Pos18"
      TagStructureMember "Position"
      TagStructureMember "Speed"
      TagStructureMember "Reached"
    TagStructureMember "Pos19"
      TagStructureMember "Position"
      TagStructureMember "Speed"
      TagStructureMember "Reached"
    TagStructureMember "Pos20"
      TagStructureMember "Position"
      TagStructureMember "Speed"
      TagStructureMember "Reached"
    TagStructureMember "Pos21"
      TagStructureMember "Position"
      TagStructureMember "Speed"
      TagStructureMember "Reached"
    TagStructureMember "Pos22"
      TagStructureMember "Position"
      TagStructureMember "Speed"
      TagStructureMember "Reached"
    TagStructureMember "Pos23"
      TagStructureMember "Position"
      TagStructureMember "Speed"
      TagStructureMember "Reached"
    TagStructureMember "Pos24"
      TagStructureMember "Position"
      TagStructureMember "Speed"
      TagStructureMember "Reached"
    TagStructureMember "Pos25"
      TagStructureMember "Position"
      TagStructureMember "Speed"
      TagStructureMember "Reached"
    TagStructureMember "Pos26"
      TagStructureMember "Position"
      TagStructureMember "Speed"
      TagStructureMember "Reached"
    TagStructureMember "Pos27"
      TagStructureMember "Position"
      TagStructureMember "Speed"
      TagStructureMember "Reached"
    TagStructureMember "Pos28"
      TagStructureMember "Position"
      TagStructureMember "Speed"
      TagStructureMember "Reached"
    TagStructureMember "Pos29"
      TagStructureMember "Position"
      TagStructureMember "Speed"
      TagStructureMember "Reached"
    TagStructureMember "Pos30"
      TagStructureMember "Position"
      TagStructureMember "Speed"
      TagStructureMember "Reached"
  Parameter_AxisRun_Axis{14} : ServoType_UDT  (PLC tag Parameter.AxisRun.Axis[14], CPU S71500-2PN_TP700, 1 s)
    TagStructureMember "Pos1"
      TagStructureMember "Position"
      TagStructureMember "Speed"
      TagStructureMember "Reached"
    TagStructureMember "Pos2"
      TagStructureMember "Position"
      TagStructureMember "Speed"
      TagStructureMember "Reached"
    TagStructureMember "Pos3"
      TagStructureMember "Position"
      TagStructureMember "Speed"
      TagStructureMember "Reached"
    TagStructureMember "Pos4"
      TagStructureMember "Position"
      TagStructureMember "Speed"
      TagStructureMember "Reached"
    TagStructureMember "Pos5"
      TagStructureMember "Position"
      TagStructureMember "Speed"
      TagStructureMember "Reached"
    TagStructureMember "Pos6"
      TagStructureMember "Position"
      TagStructureMember "Speed"
      TagStructureMember "Reached"
    TagStructureMember "Pos7"
      TagStructureMember "Position"
      TagStructureMember "Speed"
      TagStructureMember "Reached"
    TagStructureMember "Pos8"
      TagStructureMember "Position"
      TagStructureMember "Speed"
      TagStructureMember "Reached"
    TagStructureMember "Pos9"
      TagStructureMember "Position"
      TagStructureMember "Speed"
      TagStructureMember "Reached"
    TagStructureMember "Pos10"
      TagStructureMember "Position"
      TagStructureMember "Speed"
      TagStructureMember "Reached"
    TagStructureMember "Pos11"
      TagStructureMember "Position"
      TagStructureMember "Speed"
      TagStructureMember "Reached"
    TagStructureMember "Pos12"
      TagStructureMember "Position"
      TagStructureMember "Speed"
      TagStructureMember "Reached"
    TagStructureMember "Pos13"
      TagStructureMember "Position"
      TagStructureMember "Speed"
      TagStructureMember "Reached"
    TagStructureMember "Pos14"
      TagStructureMember "Position"
      TagStructureMember "Speed"
      TagStructureMember "Reached"
    TagStructureMember "Pos15"
      TagStructureMember "Position"
      TagStructureMember "Speed"
      TagStructureMember "Reached"
    TagStructureMember "Pos16"
      TagStructureMember "Position"
      TagStructureMember "Speed"
      TagStructureMember "Reached"
    TagStructureMember "Pos17"
      TagStructureMember "Position"
      TagStructureMember "Speed"
      TagStructureMember "Reached"
    TagStructureMember "Pos18"
      TagStructureMember "Position"
      TagStructureMember "Speed"
      TagStructureMember "Reached"
    TagStructureMember "Pos19"
      TagStructureMember "Position"
      TagStructureMember "Speed"
      TagStructureMember "Reached"
    TagStructureMember "Pos20"
      TagStructureMember "Position"
      TagStructureMember "Speed"
      TagStructureMember "Reached"
    TagStructureMember "Pos21"
      TagStructureMember "Position"
      TagStructureMember "Speed"
      TagStructureMember "Reached"
    TagStructureMember "Pos22"
      TagStructureMember "Position"
      TagStructureMember "Speed"
      TagStructureMember "Reached"
    TagStructureMember "Pos23"
      TagStructureMember "Position"
      TagStructureMember "Speed"
      TagStructureMember "Reached"
    TagStructureMember "Pos24"
      TagStructureMember "Position"
      TagStructureMember "Speed"
      TagStructureMember "Reached"
    TagStructureMember "Pos25"
      TagStructureMember "Position"
      TagStructureMember "Speed"
      TagStructureMember "Reached"
    TagStructureMember "Pos26"
      TagStructureMember "Position"
      TagStructureMember "Speed"
      TagStructureMember "Reached"
    TagStructureMember "Pos27"
      TagStructureMember "Position"
      TagStructureMember "Speed"
      TagStructureMember "Reached"
    TagStructureMember "Pos28"
      TagStructureMember "Position"
      TagStructureMember "Speed"
      TagStructureMember "Reached"
    TagStructureMember "Pos29"
      TagStructureMember "Position"
      TagStructureMember "Speed"
      TagStructureMember "Reached"
    TagStructureMember "Pos30"
      TagStructureMember "Position"
      TagStructureMember "Speed"
      TagStructureMember "Reached"
  Parameter_AxisRun_Axis{15} : ServoType_UDT  (PLC tag Parameter.AxisRun.Axis[15], CPU S71500-2PN_TP700, 1 s)
    TagStructureMember "Pos1"
      TagStructureMember "Position"
      TagStructureMember "Speed"
      TagStructureMember "Reached"
    TagStructureMember "Pos2"
      TagStructureMember "Position"
      TagStructureMember "Speed"
      TagStructureMember "Reached"
    TagStructureMember "Pos3"
      TagStructureMember "Position"
      TagStructureMember "Speed"
      TagStructureMember "Reached"
    TagStructureMember "Pos4"
      TagStructureMember "Position"
      TagStructureMember "Speed"
      TagStructureMember "Reached"
    TagStructureMember "Pos5"
      TagStructureMember "Position"
      TagStructureMember "Speed"
      TagStructureMember "Reached"
    TagStructureMember "Pos6"
      TagStructureMember "Position"
      TagStructureMember "Speed"
      TagStructureMember "Reached"
    TagStructureMember "Pos7"
      TagStructureMember "Position"
      TagStructureMember "Speed"
      TagStructureMember "Reached"
    TagStructureMember "Pos8"
      TagStructureMember "Position"
      TagStructureMember "Speed"
      TagStructureMember "Reached"
    TagStructureMember "Pos9"
      TagStructureMember "Position"
      TagStructureMember "Speed"
      TagStructureMember "Reached"
    TagStructureMember "Pos10"
      TagStructureMember "Position"
      TagStructureMember "Speed"
      TagStructureMember "Reached"
    TagStructureMember "Pos11"
      TagStructureMember "Position"
      TagStructureMember "Speed"
      TagStructureMember "Reached"
    TagStructureMember "Pos12"
      TagStructureMember "Position"
      TagStructureMember "Speed"
      TagStructureMember "Reached"
    TagStructureMember "Pos13"
      TagStructureMember "Position"
      TagStructureMember "Speed"
      TagStructureMember "Reached"
    TagStructureMember "Pos14"
      TagStructureMember "Position"
      TagStructureMember "Speed"
      TagStructureMember "Reached"
    TagStructureMember "Pos15"
      TagStructureMember "Position"
      TagStructureMember "Speed"
      TagStructureMember "Reached"
    TagStructureMember "Pos16"
      TagStructureMember "Position"
      TagStructureMember "Speed"
      TagStructureMember "Reached"
    TagStructureMember "Pos17"
      TagStructureMember "Position"
      TagStructureMember "Speed"
      TagStructureMember "Reached"
    TagStructureMember "Pos18"
      TagStructureMember "Position"
      TagStructureMember "Speed"
      TagStructureMember "Reached"
    TagStructureMember "Pos19"
      TagStructureMember "Position"
      TagStructureMember "Speed"
      TagStructureMember "Reached"
    TagStructureMember "Pos20"
      TagStructureMember "Position"
      TagStructureMember "Speed"
      TagStructureMember "Reached"
    TagStructureMember "Pos21"
      TagStructureMember "Position"
      TagStructureMember "Speed"
      TagStructureMember "Reached"
    TagStructureMember "Pos22"
      TagStructureMember "Position"
      TagStructureMember "Speed"
      TagStructureMember "Reached"
    TagStructureMember "Pos23"
      TagStructureMember "Position"
      TagStructureMember "Speed"
      TagStructureMember "Reached"
    TagStructureMember "Pos24"
      TagStructureMember "Position"
      TagStructureMember "Speed"
      TagStructureMember "Reached"
    TagStructureMember "Pos25"
      TagStructureMember "Position"
      TagStructureMember "Speed"
      TagStructureMember "Reached"
    TagStructureMember "Pos26"
      TagStructureMember "Position"
      TagStructureMember "Speed"
      TagStructureMember "Reached"
    TagStructureMember "Pos27"
      TagStructureMember "Position"
      TagStructureMember "Speed"
      TagStructureMember "Reached"
    TagStructureMember "Pos28"
      TagStructureMember "Position"
      TagStructureMember "Speed"
      TagStructureMember "Reached"
    TagStructureMember "Pos29"
      TagStructureMember "Position"
      TagStructureMember "Speed"
      TagStructureMember "Reached"
    TagStructureMember "Pos30"
      TagStructureMember "Position"
      TagStructureMember "Speed"
      TagStructureMember "Reached"
